TYPE LAxisCtrl_typeStop :
STRUCT

	deceleration		: LREAL;
	jerk				: REAL;
	abortAcceleration	: BOOL;

END_STRUCT
END_TYPE

(* stored: Version 1.1.0.1
   DUT LAxisCtrl_typeStop: Id {fbf51fd2-0703-4d04-8a18-c9e424616f8c} *)
